// TIA Portal project "Cuối kì" (V16)

(* hardware
DEVICE "S7-1200 station_1"  S7-1200 Station
   slot 0: "Rack_0"  S7-1200 Rack  Rack  V1.0
   slot 1: "PLC_1"  CPU 1212C DC/DC/DC  6ES7 212-1AE40-0XB0  V4.4
*)

// ===== PLC "PLC_1"  CPU 1212C DC/DC/DC =====

VAR_GLOBAL   // PLC tag table "Default tag table"
   "Clock_Byte" AT %MB21 : Byte;
   "Clock_10Hz" AT %M21.0 : Bool;
   "Clock_5Hz" AT %M21.1 : Bool;
   "Clock_2.5Hz" AT %M21.2 : Bool;
   "Clock_2Hz" AT %M21.3 : Bool;
   "Clock_1.25Hz" AT %M21.4 : Bool;
   "Clock_1Hz" AT %M21.5 : Bool;
   "Clock_0.625Hz" AT %M21.6 : Bool;
   "Clock_0.5Hz" AT %M21.7 : Bool;
   "iStart" AT %M0.0 : Bool;
   "iStop" AT %M0.1 : Bool;
   "enableSystem" AT %M0.2 : Bool;
   "mEnableXiloRice" AT %M0.3 : Bool;
   "mEnableXiloCorn" AT %M0.4 : Bool;
   "mEnableXiloManioc" AT %M0.5 : Bool;
   "mEnableXiloBean" AT %M0.6 : Bool;
   "mEnableXiloFish" AT %M0.7 : Bool;
   "mLetOutRice" AT %M1.0 : Bool;
   "mLetOutCorn" AT %M1.1 : Bool;
   "mLetOutManioc" AT %M1.2 : Bool;
   "mLetOutBean" AT %M1.3 : Bool;
   "mLetOutFish" AT %M1.4 : Bool;
   "mLightRice" AT %M1.5 : Bool;
   "mLightCorn" AT %M1.6 : Bool;
   "mLightManioc" AT %M1.7 : Bool;
   "mLightBean" AT %M2.0 : Bool;
   "mLightFish" AT %M2.1 : Bool;
   "iResetCTU" AT %M2.2 : Bool;
   "oXilo1" AT %Q0.0 : Bool;
   "oXilo2" AT %Q0.1 : Bool;
   "oXilo3" AT %Q0.2 : Bool;
   "oXilo4" AT %Q0.3 : Bool;
   "oXilo5" AT %Q0.4 : Bool;
   "oXilo6" AT %Q0.5 : Bool;
   "oXilo7" AT %Q0.6 : Bool;
   "oXilo8" AT %Q0.7 : Bool;
   "oXilo9" AT %Q1.0 : Bool;
   "oXilo10" AT %Q1.1 : Bool;
   "oXilo11" AT %Q1.2 : Bool;
   "oXilo12" AT %Q1.3 : Bool;
   "oXilo13" AT %Q1.4 : Bool;
   "oXilo14" AT %Q1.5 : Bool;
   "oXilo15" AT %Q1.6 : Bool;
   "oXilo16" AT %Q1.7 : Bool;
   "mLetOutScale" AT %M2.3 : Bool;
   "iSensor1" AT %M2.4 : Bool;
   "iSensorHigh2" AT %M2.5 : Bool;
   "iSensorLow2" AT %M2.6 : Bool;
   "oValve1" AT %Q2.0 : Bool;
   "oValve2" AT %Q2.1 : Bool;
   "iResetCTD" AT %M2.7 : Bool;
   "mTank" AT %M3.0 : Bool;
   "Tag_3" AT %M100.1 : Bool;
   "Tag_4" AT %M100.2 : Bool;
   "oMix" AT %Q2.2 : Bool;
   "iContinue" AT %M3.1 : Bool;
   "Continue" AT %M3.2 : Bool;
   "oValve3" AT %Q2.3 : Bool;
   "iSensor3" AT %M3.4 : Bool;
   "Hold11" AT %M3.6 : Bool;
   "Hold21" AT %M3.7 : Bool;
   "Hold31" AT %M4.0 : Bool;
   "Hold41" AT %M4.1 : Bool;
   "Hold51" AT %M4.2 : Bool;
   "Reset" AT %M4.3 : Bool;
   "Hold12" AT %M4.4 : Bool;
   "Hold13" AT %M4.5 : Bool;
   "Hold14" AT %M4.6 : Bool;
   "Hold15" AT %M4.7 : Bool;
   "Hold22" AT %M5.0 : Bool;
   "Hold23" AT %M5.1 : Bool;
   "Hold24" AT %M5.2 : Bool;
   "Hold25" AT %M5.3 : Bool;
   "Hold32" AT %M5.4 : Bool;
   "Hold33" AT %M5.5 : Bool;
   "Hold34" AT %M5.6 : Bool;
   "Hold35" AT %M5.7 : Bool;
   "Hold42" AT %M6.0 : Bool;
   "Hold52" AT %M6.1 : Bool;
   "Tag_1" AT %MW1 : Int;
   "Tag_2" AT %MW2 : Int;
   "Tag_5" AT %MW3 : Int;
   "Tag_6" AT %MW4 : Int;
   "Tag_7" AT %MW5 : Int;
   "Tag_8" AT %MW6 : Int;
   "Tag_9" AT %MW7 : Int;
   "Tag_10" AT %MW8 : Int;
   "Tag_11" AT %MW9 : Int;
   "Tag_12" AT %MW10 : Int;
   "Tag_13" AT %MW11 : Int;
   "Tag_14" AT %MW12 : Int;
   "Tag_15" AT %MW13 : Int;
   "Tag_16" AT %MW14 : Int;
   "Tag_17" AT %MW15 : Int;
   "Tag_18" AT %MW16 : Int;
   "Tag_19" AT %MW17 : Int;
   "Tag_20" AT %MW18 : Int;
   "Tag_21" AT %MD1 : Time;
   "oSensor1" AT %M6.2 : Bool;
   "oSensor3" AT %M6.3 : Bool;
END_VAR

DATA_BLOCK "Mass"   // DB1
{ S7_Optimized_Access := 'FALSE' }
VERSION : 0.1
   VAR
      Rice : Int := 5;
      Corn : Int := 5;
      Manioc : Int := 5;
      Bean : Int := 5;
      Fish : Int := 5;
   END_VAR
BEGIN
END_DATA_BLOCK

DATA_BLOCK "TimeMix"   // DB2
{ S7_Optimized_Access := 'FALSE' }
VERSION : 0.1
   VAR
      "Time" : Time := T#40S;
   END_VAR
BEGIN
END_DATA_BLOCK

DATA_BLOCK "Sum"   // DB22
{ S7_Optimized_Access := 'FALSE' }
VERSION : 0.1
   VAR
      Rice : Int := 60;
      Corn : Int := 50;
      Manioc : Int := 60;
      Bean : Int := 30;
      Fish : Int := 60;
      Sum1 : Int := 100;
      Sum2 : Int := 200;
   END_VAR
BEGIN
END_DATA_BLOCK

DATA_BLOCK "Weight"   // DB23
{ S7_Optimized_Access := 'FALSE' }
VERSION : 0.1
   VAR
      Xilo1 : Int;
      Xilo2 : Int;
      Xilo3 : Int;
      Xilo4 : Int;
      Xilo5 : Int;
      Xilo6 : Int;
      Xilo7 : Int;
      Xilo8 : Int;
      Xilo9 : Int;
      Xilo10 : Int;
      Xilo11 : Int;
      Xilo12 : Int;
      Xilo13 : Int;
      Xilo14 : Int;
      Xilo15 : Int;
      Xilo16 : Int;
      Sum1 : Int;
      Sum2 : Int;
   END_VAR
BEGIN
END_DATA_BLOCK

DATA_BLOCK "ADD"   // DB24
{ S7_Optimized_Access := 'FALSE' }
VERSION : 0.1
   VAR
      ScaleSum1 : Int;
      ScaleSum2 : Int;
   END_VAR
BEGIN
END_DATA_BLOCK

// folder: System blocks/Program resources

DATA_BLOCK "Scale8"   // DB3
{ S7_Optimized_Access := 'TRUE' }
AUTHOR : Simatic
FAMILY : IEC
NAME : CNTR
VERSION : 1.0
// stored: InstanceOfName IEC_COUNTER
"IEC_COUNTER"
BEGIN
END_DATA_BLOCK

DATA_BLOCK "Scale9"   // DB4
{ S7_Optimized_Access := 'TRUE' }
AUTHOR : Simatic
FAMILY : IEC
NAME : CNTR
VERSION : 1.0
// stored: InstanceOfName IEC_COUNTER
"IEC_COUNTER"
BEGIN
END_DATA_BLOCK

DATA_BLOCK "Scale4"   // DB5
{ S7_Optimized_Access := 'TRUE' }
AUTHOR : Simatic
FAMILY : IEC
NAME : CNTR
VERSION : 1.0
// stored: InstanceOfName IEC_COUNTER
"IEC_COUNTER"
BEGIN
END_DATA_BLOCK

DATA_BLOCK "Scale5"   // DB6
{ S7_Optimized_Access := 'TRUE' }
AUTHOR : Simatic
FAMILY : IEC
NAME : CNTR
VERSION : 1.0
// stored: InstanceOfName IEC_COUNTER
"IEC_COUNTER"
BEGIN
END_DATA_BLOCK

DATA_BLOCK "Scale6"   // DB7
{ S7_Optimized_Access := 'TRUE' }
AUTHOR : Simatic
FAMILY : IEC
NAME : CNTR
VERSION : 1.0
// stored: InstanceOfName IEC_COUNTER
"IEC_COUNTER"
BEGIN
END_DATA_BLOCK

DATA_BLOCK "Scale7"   // DB8
{ S7_Optimized_Access := 'TRUE' }
AUTHOR : Simatic
FAMILY : IEC
NAME : CNTR
VERSION : 1.0
// stored: InstanceOfName IEC_COUNTER
"IEC_COUNTER"
BEGIN
END_DATA_BLOCK

DATA_BLOCK "Scale1"   // DB9
{ S7_Optimized_Access := 'TRUE' }
AUTHOR : Simatic
FAMILY : IEC
NAME : CNTR
VERSION : 1.0
// stored: InstanceOfName IEC_COUNTER
"IEC_COUNTER"
BEGIN
END_DATA_BLOCK

DATA_BLOCK "Scale2"   // DB10
{ S7_Optimized_Access := 'TRUE' }
AUTHOR : Simatic
FAMILY : IEC
NAME : CNTR
VERSION : 1.0
// stored: InstanceOfName IEC_COUNTER
"IEC_COUNTER"
BEGIN
END_DATA_BLOCK

DATA_BLOCK "Scale3"   // DB11
{ S7_Optimized_Access := 'TRUE' }
AUTHOR : Simatic
FAMILY : IEC
NAME : CNTR
VERSION : 1.0
// stored: InstanceOfName IEC_COUNTER
"IEC_COUNTER"
BEGIN
END_DATA_BLOCK

DATA_BLOCK "Scale10"   // DB12
{ S7_Optimized_Access := 'TRUE' }
AUTHOR : Simatic
FAMILY : IEC
NAME : CNTR
VERSION : 1.0
// stored: InstanceOfName IEC_COUNTER
"IEC_COUNTER"
BEGIN
END_DATA_BLOCK

DATA_BLOCK "Scale11"   // DB13
{ S7_Optimized_Access := 'TRUE' }
AUTHOR : Simatic
FAMILY : IEC
NAME : CNTR
VERSION : 1.0
// stored: InstanceOfName IEC_COUNTER
"IEC_COUNTER"
BEGIN
END_DATA_BLOCK

DATA_BLOCK "Scale12"   // DB14
{ S7_Optimized_Access := 'TRUE' }
AUTHOR : Simatic
FAMILY : IEC
NAME : CNTR
VERSION : 1.0
// stored: InstanceOfName IEC_COUNTER
"IEC_COUNTER"
BEGIN
END_DATA_BLOCK

DATA_BLOCK "Scale13"   // DB15
{ S7_Optimized_Access := 'TRUE' }
AUTHOR : Simatic
FAMILY : IEC
NAME : CNTR
VERSION : 1.0
// stored: InstanceOfName IEC_COUNTER
"IEC_COUNTER"
BEGIN
END_DATA_BLOCK

DATA_BLOCK "Scale14"   // DB16
{ S7_Optimized_Access := 'TRUE' }
AUTHOR : Simatic
FAMILY : IEC
NAME : CNTR
VERSION : 1.0
// stored: InstanceOfName IEC_COUNTER
"IEC_COUNTER"
BEGIN
END_DATA_BLOCK

DATA_BLOCK "Scale15"   // DB17
{ S7_Optimized_Access := 'TRUE' }
AUTHOR : Simatic
FAMILY : IEC
NAME : CNTR
VERSION : 1.0
// stored: InstanceOfName IEC_COUNTER
"IEC_COUNTER"
BEGIN
END_DATA_BLOCK

DATA_BLOCK "Scale16"   // DB18
{ S7_Optimized_Access := 'TRUE' }
AUTHOR : Simatic
FAMILY : IEC
NAME : CNTR
VERSION : 1.0
// stored: InstanceOfName IEC_COUNTER
"IEC_COUNTER"
BEGIN
END_DATA_BLOCK

DATA_BLOCK "ScaleSum"   // DB19
{ S7_Optimized_Access := 'TRUE' }
AUTHOR : Simatic
FAMILY : IEC
NAME : CNTR
VERSION : 1.0
// stored: InstanceOfName IEC_COUNTER
"IEC_COUNTER"
BEGIN
END_DATA_BLOCK

DATA_BLOCK "Time"   // DB20
{ S7_Optimized_Access := 'TRUE' }
AUTHOR : Simatic
FAMILY : IEC
NAME : IEC_TMR
VERSION : 1.0
// stored: InstanceOfName IEC_TIMER
"IEC_TIMER"
BEGIN
END_DATA_BLOCK

DATA_BLOCK "ScaleSum2"   // DB21
{ S7_Optimized_Access := 'TRUE' }
AUTHOR : Simatic
FAMILY : IEC
NAME : CNTR
VERSION : 1.0
// stored: InstanceOfName IEC_COUNTER
"IEC_COUNTER"
BEGIN
END_DATA_BLOCK

// folder: (top level)

ORGANIZATION_BLOCK "Main"   // OB1, LAD, ProgramCycle
TITLE = "Main Program Sweep (Cycle)"
{ S7_Optimized_Access := 'TRUE' }
VERSION : 0.1
   VAR_INPUT
      Initial_Call : Bool;   // Initial call of this OB
      Remanence : Bool;   // =True, if remanent data are available
   END_VAR
   VAR_TEMP   // added for the SCL form of the ladder/FBD networks
      _w1 : Bool;
      _w2 : Bool;
      _w3 : Bool;
   END_VAR
BEGIN

REGION Network 1: Open/Close System
   // Bắt đầu + đóng + tiếp tục + reset counter
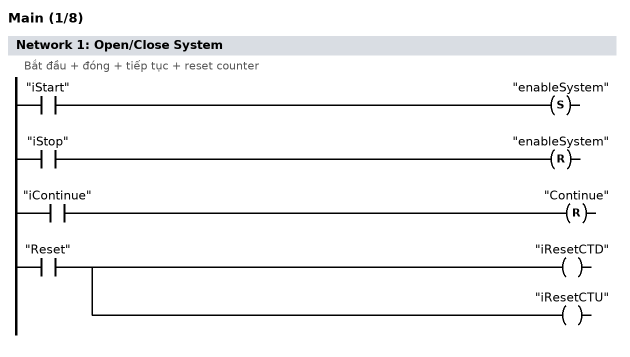
   RUNG wire#powerrail
      Contact( "iStart" )
      S_Coil( "enableSystem" )
   END_RUNG
   RUNG wire#powerrail
      Contact( "iStop" )
      R_Coil( "enableSystem" )
   END_RUNG
   RUNG wire#powerrail
      Contact( "iContinue" )
      R_Coil( "Continue" )
   END_RUNG
   RUNG wire#powerrail
      Contact( "Reset" )
      wire#w1
      Coil( "iResetCTD" )
   END_RUNG
   RUNG wire#w1
      Coil( "iResetCTU" )
   END_RUNG
   // the same network as SCL:
   IF "iStart" THEN "enableSystem" := TRUE; END_IF;
   IF "iStop" THEN "enableSystem" := FALSE; END_IF;
   IF "iContinue" THEN "Continue" := FALSE; END_IF;
   "iResetCTD" := "Reset";
   "iResetCTU" := "Reset";
END_REGION

REGION Network 2: So sánh khối lượng
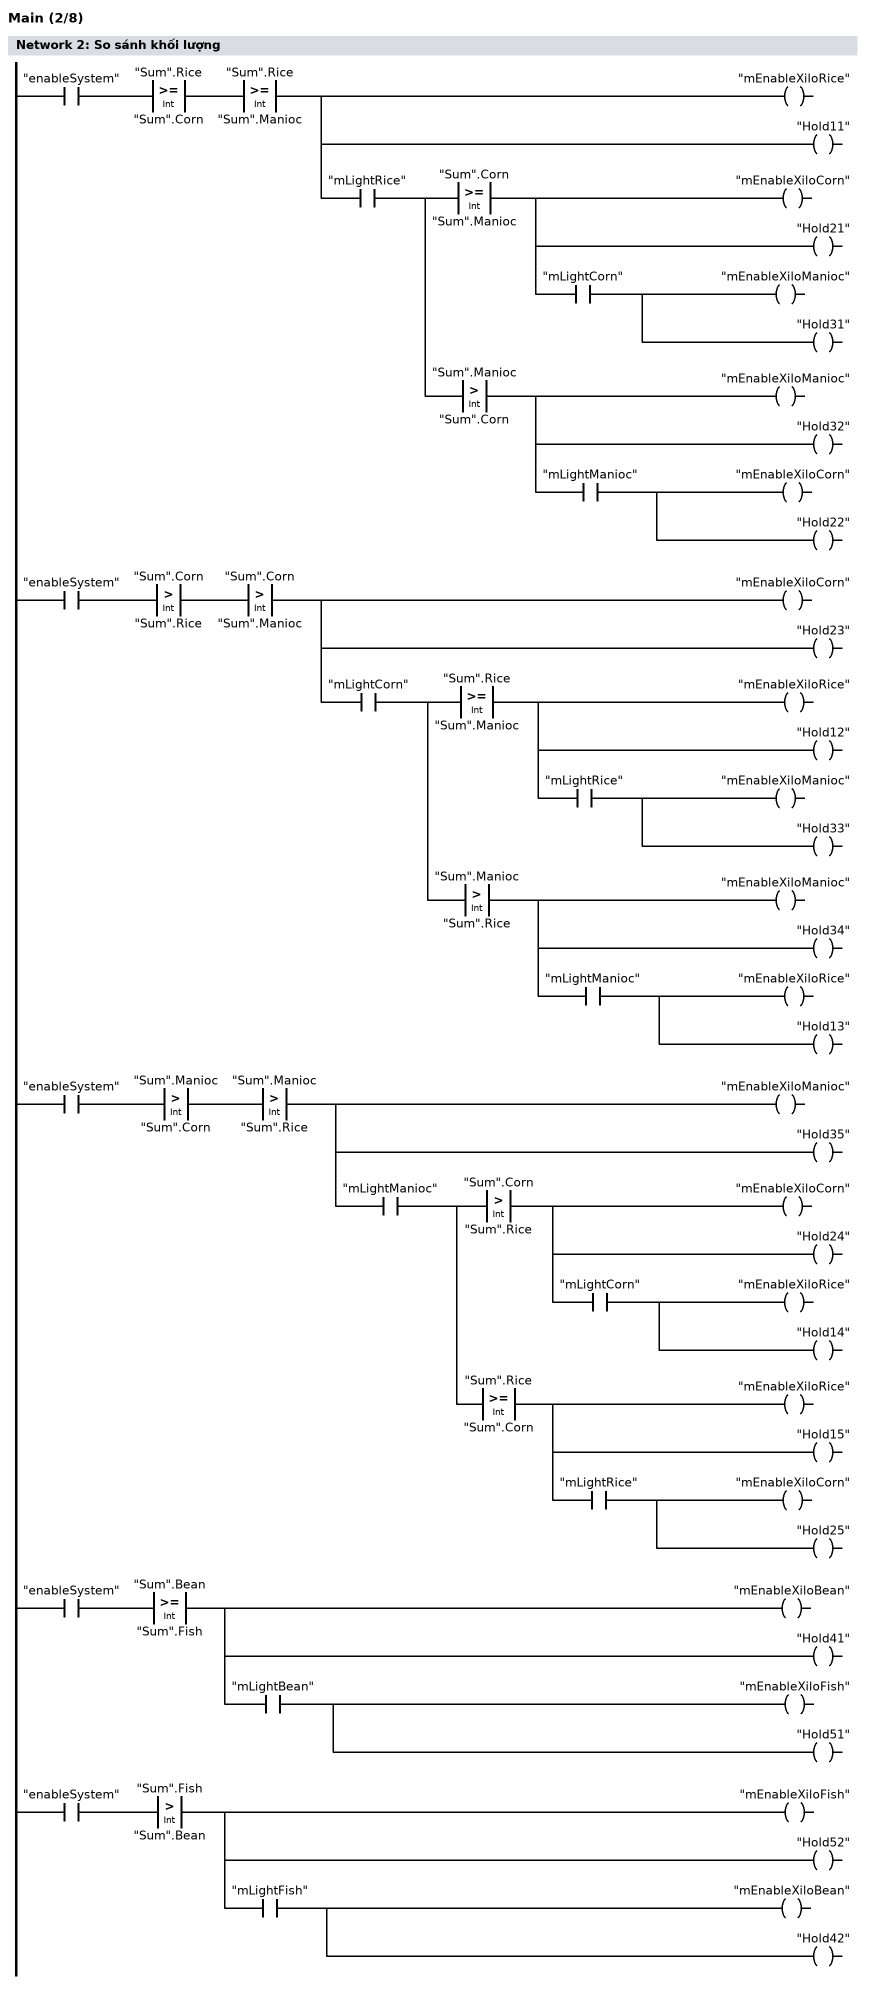
   RUNG wire#powerrail
      Contact( "enableSystem" )
      { S7_Templates := "SrcType := Int" } GE_Contact(in1 := "Sum".Rice, in2 := "Sum".Corn)
      { S7_Templates := "SrcType := Int" } GE_Contact(in1 := "Sum".Rice, in2 := "Sum".Manioc)
      wire#w1
      Coil( "mEnableXiloRice" )
   END_RUNG
   RUNG wire#w1
      Coil( "Hold11" )
   END_RUNG
   RUNG wire#w1
      Contact( "mLightRice" )
      wire#w2
      { S7_Templates := "SrcType := Int" } GE_Contact(in1 := "Sum".Corn, in2 := "Sum".Manioc)
      wire#w3
      Coil( "mEnableXiloCorn" )
   END_RUNG
   RUNG wire#w3
      Coil( "Hold21" )
   END_RUNG
   RUNG wire#w3
      Contact( "mLightCorn" )
      wire#w4
      Coil( "mEnableXiloManioc" )
   END_RUNG
   RUNG wire#w4
      Coil( "Hold31" )
   END_RUNG
   RUNG wire#w2
      { S7_Templates := "SrcType := Int" } GT_Contact(in1 := "Sum".Manioc, in2 := "Sum".Corn)
      wire#w5
      Coil( "mEnableXiloManioc" )
   END_RUNG
   RUNG wire#w5
      Coil( "Hold32" )
   END_RUNG
   RUNG wire#w5
      Contact( "mLightManioc" )
      wire#w6
      Coil( "mEnableXiloCorn" )
   END_RUNG
   RUNG wire#w6
      Coil( "Hold22" )
   END_RUNG
   RUNG wire#powerrail
      Contact( "enableSystem" )
      { S7_Templates := "SrcType := Int" } GT_Contact(in1 := "Sum".Corn, in2 := "Sum".Rice)
      { S7_Templates := "SrcType := Int" } GT_Contact(in1 := "Sum".Corn, in2 := "Sum".Manioc)
      wire#w7
      Coil( "mEnableXiloCorn" )
   END_RUNG
   RUNG wire#w7
      Coil( "Hold23" )
   END_RUNG
   RUNG wire#w7
      Contact( "mLightCorn" )
      wire#w8
      { S7_Templates := "SrcType := Int" } GE_Contact(in1 := "Sum".Rice, in2 := "Sum".Manioc)
      wire#w9
      Coil( "mEnableXiloRice" )
   END_RUNG
   RUNG wire#w9
      Coil( "Hold12" )
   END_RUNG
   RUNG wire#w9
      Contact( "mLightRice" )
      wire#w10
      Coil( "mEnableXiloManioc" )
   END_RUNG
   RUNG wire#w10
      Coil( "Hold33" )
   END_RUNG
   RUNG wire#w8
      { S7_Templates := "SrcType := Int" } GT_Contact(in1 := "Sum".Manioc, in2 := "Sum".Rice)
      wire#w11
      Coil( "mEnableXiloManioc" )
   END_RUNG
   RUNG wire#w11
      Coil( "Hold34" )
   END_RUNG
   RUNG wire#w11
      Contact( "mLightManioc" )
      wire#w12
      Coil( "mEnableXiloRice" )
   END_RUNG
   RUNG wire#w12
      Coil( "Hold13" )
   END_RUNG
   RUNG wire#powerrail
      Contact( "enableSystem" )
      { S7_Templates := "SrcType := Int" } GT_Contact(in1 := "Sum".Manioc, in2 := "Sum".Corn)
      { S7_Templates := "SrcType := Int" } GT_Contact(in1 := "Sum".Manioc, in2 := "Sum".Rice)
      wire#w13
      Coil( "mEnableXiloManioc" )
   END_RUNG
   RUNG wire#w13
      Coil( "Hold35" )
   END_RUNG
   RUNG wire#w13
      Contact( "mLightManioc" )
      wire#w14
      { S7_Templates := "SrcType := Int" } GT_Contact(in1 := "Sum".Corn, in2 := "Sum".Rice)
      wire#w15
      Coil( "mEnableXiloCorn" )
   END_RUNG
   RUNG wire#w15
      Coil( "Hold24" )
   END_RUNG
   RUNG wire#w15
      Contact( "mLightCorn" )
      wire#w16
      Coil( "mEnableXiloRice" )
   END_RUNG
   RUNG wire#w16
      Coil( "Hold14" )
   END_RUNG
   RUNG wire#w14
      { S7_Templates := "SrcType := Int" } GE_Contact(in1 := "Sum".Rice, in2 := "Sum".Corn)
      wire#w17
      Coil( "mEnableXiloRice" )
   END_RUNG
   RUNG wire#w17
      Coil( "Hold15" )
   END_RUNG
   RUNG wire#w17
      Contact( "mLightRice" )
      wire#w18
      Coil( "mEnableXiloCorn" )
   END_RUNG
   RUNG wire#w18
      Coil( "Hold25" )
   END_RUNG
   RUNG wire#powerrail
      Contact( "enableSystem" )
      { S7_Templates := "SrcType := Int" } GE_Contact(in1 := "Sum".Bean, in2 := "Sum".Fish)
      wire#w19
      Coil( "mEnableXiloBean" )
   END_RUNG
   RUNG wire#w19
      Coil( "Hold41" )
   END_RUNG
   RUNG wire#w19
      Contact( "mLightBean" )
      wire#w20
      Coil( "mEnableXiloFish" )
   END_RUNG
   RUNG wire#w20
      Coil( "Hold51" )
   END_RUNG
   RUNG wire#powerrail
      Contact( "enableSystem" )
      { S7_Templates := "SrcType := Int" } GT_Contact(in1 := "Sum".Fish, in2 := "Sum".Bean)
      wire#w21
      Coil( "mEnableXiloFish" )
   END_RUNG
   RUNG wire#w21
      Coil( "Hold52" )
   END_RUNG
   RUNG wire#w21
      Contact( "mLightFish" )
      wire#w22
      Coil( "mEnableXiloBean" )
   END_RUNG
   RUNG wire#w22
      Coil( "Hold42" )
   END_RUNG
   // the same network as SCL:
   "mEnableXiloRice" := "enableSystem" AND ("Sum".Rice >= "Sum".Corn) AND ("Sum".Rice >= "Sum".Manioc);
   "Hold11" := "mEnableXiloRice";
   #_w1 := "mEnableXiloRice" AND "mLightRice";
   "mEnableXiloCorn" := #_w1 AND ("Sum".Corn >= "Sum".Manioc);
   "Hold21" := "mEnableXiloCorn";
   "mEnableXiloManioc" := "mEnableXiloCorn" AND "mLightCorn";
   "Hold31" := "mEnableXiloManioc";
   "mEnableXiloManioc" := #_w1 AND ("Sum".Manioc > "Sum".Corn);
   "Hold32" := "mEnableXiloManioc";
   "mEnableXiloCorn" := "mEnableXiloManioc" AND "mLightManioc";
   "Hold22" := "mEnableXiloCorn";
   "mEnableXiloCorn" := "enableSystem" AND ("Sum".Corn > "Sum".Rice) AND ("Sum".Corn > "Sum".Manioc);
   "Hold23" := "mEnableXiloCorn";
   #_w2 := "mEnableXiloCorn" AND "mLightCorn";
   "mEnableXiloRice" := #_w2 AND ("Sum".Rice >= "Sum".Manioc);
   "Hold12" := "mEnableXiloRice";
   "mEnableXiloManioc" := "mEnableXiloRice" AND "mLightRice";
   "Hold33" := "mEnableXiloManioc";
   "mEnableXiloManioc" := #_w2 AND ("Sum".Manioc > "Sum".Rice);
   "Hold34" := "mEnableXiloManioc";
   "mEnableXiloRice" := "mEnableXiloManioc" AND "mLightManioc";
   "Hold13" := "mEnableXiloRice";
   "mEnableXiloManioc" := "enableSystem" AND ("Sum".Manioc > "Sum".Corn) AND ("Sum".Manioc > "Sum".Rice);
   "Hold35" := "mEnableXiloManioc";
   #_w3 := "mEnableXiloManioc" AND "mLightManioc";
   "mEnableXiloCorn" := #_w3 AND ("Sum".Corn > "Sum".Rice);
   "Hold24" := "mEnableXiloCorn";
   "mEnableXiloRice" := "mEnableXiloCorn" AND "mLightCorn";
   "Hold14" := "mEnableXiloRice";
   "mEnableXiloRice" := #_w3 AND ("Sum".Rice >= "Sum".Corn);
   "Hold15" := "mEnableXiloRice";
   "mEnableXiloCorn" := "mEnableXiloRice" AND "mLightRice";
   "Hold25" := "mEnableXiloCorn";
   "mEnableXiloBean" := "enableSystem" AND ("Sum".Bean >= "Sum".Fish);
   "Hold41" := "mEnableXiloBean";
   "mEnableXiloFish" := "mEnableXiloBean" AND "mLightBean";
   "Hold51" := "mEnableXiloFish";
   "mEnableXiloFish" := "enableSystem" AND ("Sum".Fish > "Sum".Bean);
   "Hold52" := "mEnableXiloFish";
   "mEnableXiloBean" := "mEnableXiloFish" AND "mLightFish";
   "Hold42" := "mEnableXiloBean";
END_REGION

REGION Network 3: Mở nguồn các xilo
   // Mở nguồn các xilo
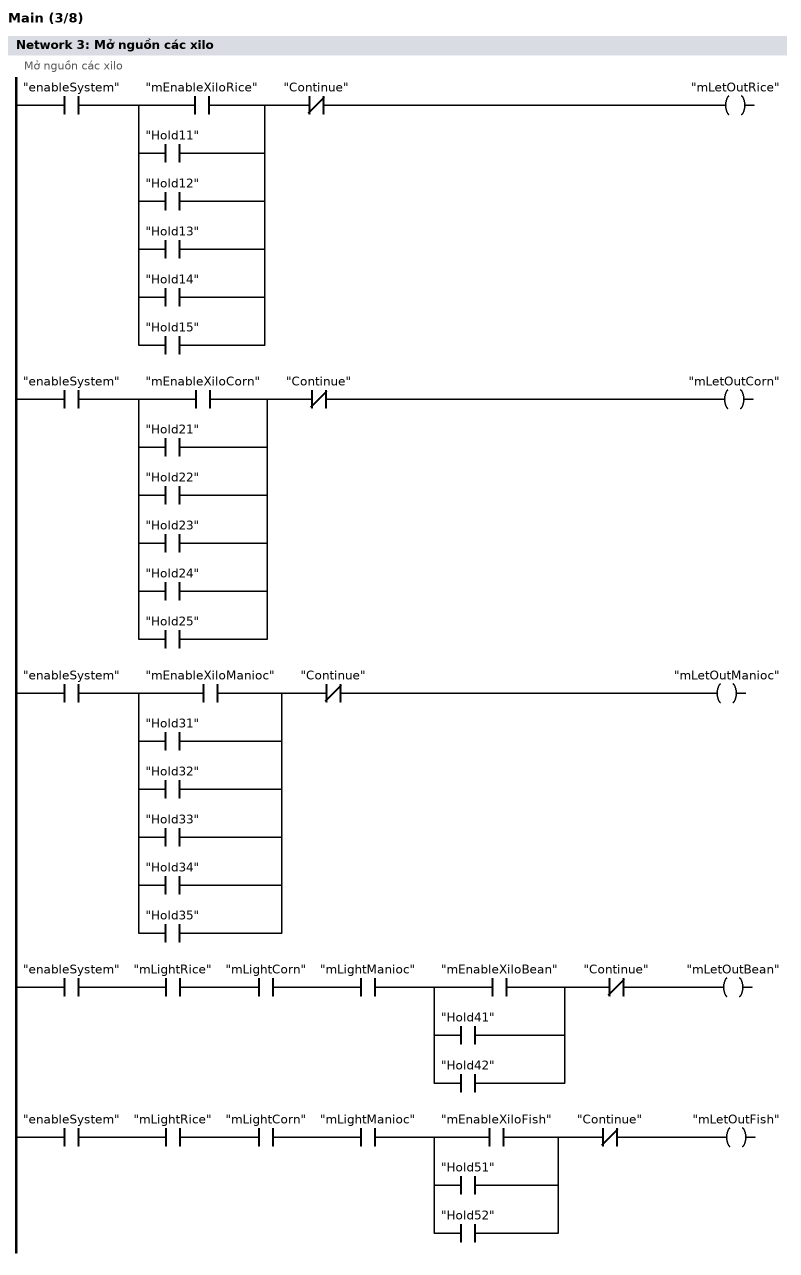
   RUNG wire#powerrail
      Contact( "enableSystem" )
      wire#w1
      Contact( "mEnableXiloRice" )
      wire#w2
      I_Contact( "Continue" )
      Coil( "mLetOutRice" )
   END_RUNG
   RUNG wire#w1
      Contact( "Hold11" )
   END_RUNG wire#w2
   RUNG wire#w1
      Contact( "Hold12" )
   END_RUNG wire#w2
   RUNG wire#w1
      Contact( "Hold13" )
   END_RUNG wire#w2
   RUNG wire#w1
      Contact( "Hold14" )
   END_RUNG wire#w2
   RUNG wire#w1
      Contact( "Hold15" )
   END_RUNG wire#w2
   RUNG wire#powerrail
      Contact( "enableSystem" )
      wire#w3
      Contact( "mEnableXiloCorn" )
      wire#w4
      I_Contact( "Continue" )
      Coil( "mLetOutCorn" )
   END_RUNG
   RUNG wire#w3
      Contact( "Hold21" )
   END_RUNG wire#w4
   RUNG wire#w3
      Contact( "Hold22" )
   END_RUNG wire#w4
   RUNG wire#w3
      Contact( "Hold23" )
   END_RUNG wire#w4
   RUNG wire#w3
      Contact( "Hold24" )
   END_RUNG wire#w4
   RUNG wire#w3
      Contact( "Hold25" )
   END_RUNG wire#w4
   RUNG wire#powerrail
      Contact( "enableSystem" )
      wire#w5
      Contact( "mEnableXiloManioc" )
      wire#w6
      I_Contact( "Continue" )
      Coil( "mLetOutManioc" )
   END_RUNG
   RUNG wire#w5
      Contact( "Hold31" )
   END_RUNG wire#w6
   RUNG wire#w5
      Contact( "Hold32" )
   END_RUNG wire#w6
   RUNG wire#w5
      Contact( "Hold33" )
   END_RUNG wire#w6
   RUNG wire#w5
      Contact( "Hold34" )
   END_RUNG wire#w6
   RUNG wire#w5
      Contact( "Hold35" )
   END_RUNG wire#w6
   RUNG wire#powerrail
      Contact( "enableSystem" )
      Contact( "mLightRice" )
      Contact( "mLightCorn" )
      Contact( "mLightManioc" )
      wire#w7
      Contact( "mEnableXiloBean" )
      wire#w8
      I_Contact( "Continue" )
      Coil( "mLetOutBean" )
   END_RUNG
   RUNG wire#w7
      Contact( "Hold41" )
   END_RUNG wire#w8
   RUNG wire#w7
      Contact( "Hold42" )
   END_RUNG wire#w8
   RUNG wire#powerrail
      Contact( "enableSystem" )
      Contact( "mLightRice" )
      Contact( "mLightCorn" )
      Contact( "mLightManioc" )
      wire#w9
      Contact( "mEnableXiloFish" )
      wire#w10
      I_Contact( "Continue" )
      Coil( "mLetOutFish" )
   END_RUNG
   RUNG wire#w9
      Contact( "Hold51" )
   END_RUNG wire#w10
   RUNG wire#w9
      Contact( "Hold52" )
   END_RUNG wire#w10
   // the same network as SCL:
   "mLetOutRice" := "enableSystem" AND ("mEnableXiloRice" OR "Hold11" OR "Hold12" OR "Hold13" OR "Hold14" OR "Hold15") AND NOT "Continue";
   "mLetOutCorn" := "enableSystem" AND ("mEnableXiloCorn" OR "Hold21" OR "Hold22" OR "Hold23" OR "Hold24" OR "Hold25") AND NOT "Continue";
   "mLetOutManioc" := "enableSystem" AND ("mEnableXiloManioc" OR "Hold31" OR "Hold32" OR "Hold33" OR "Hold34" OR "Hold35") AND NOT "Continue";
   "mLetOutBean" := "enableSystem" AND "mLightRice" AND "mLightCorn" AND "mLightManioc" AND ("mEnableXiloBean" OR "Hold41" OR "Hold42") AND NOT "Continue";
   "mLetOutFish" := "enableSystem" AND "mLightRice" AND "mLightCorn" AND "mLightManioc" AND ("mEnableXiloFish" OR "Hold51" OR "Hold52") AND NOT "Continue";
END_REGION

REGION Network 4: xả xilo 1,2,3 (bột gạo)
   // xả xilo 1,2,3 (bột gạo)
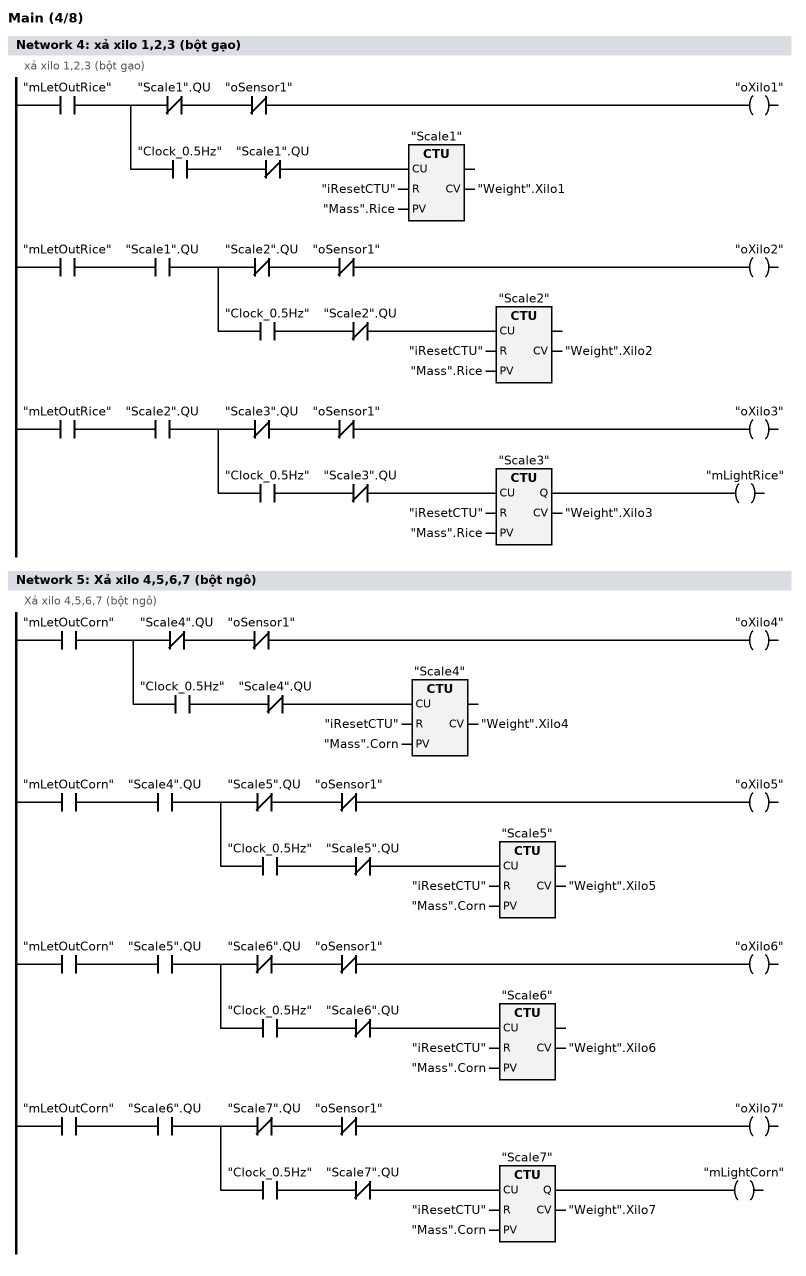
   "oXilo1" := "mLetOutRice" AND NOT "Scale1".QU AND NOT "oSensor1";
   "Scale1".CTU(CU := "mLetOutRice" AND "Clock_0.5Hz" AND NOT "Scale1".QU,
                R := "iResetCTU",
                PV := "Mass".Rice,
                CV => "Weight".Xilo1);
   #_w1 := "mLetOutRice" AND "Scale1".QU;
   "oXilo2" := #_w1 AND NOT "Scale2".QU AND NOT "oSensor1";
   "Scale2".CTU(CU := #_w1 AND "Clock_0.5Hz" AND NOT "Scale2".QU,
                R := "iResetCTU",
                PV := "Mass".Rice,
                CV => "Weight".Xilo2);
   #_w2 := "mLetOutRice" AND "Scale2".QU;
   "oXilo3" := #_w2 AND NOT "Scale3".QU AND NOT "oSensor1";
   "Scale3".CTU(CU := #_w2 AND "Clock_0.5Hz" AND NOT "Scale3".QU,
                R := "iResetCTU",
                PV := "Mass".Rice,
                CV => "Weight".Xilo3);
   "mLightRice" := "Scale3".Q;
END_REGION

REGION Network 5: Xả xilo 4,5,6,7 (bột ngô)
   // Xả xilo 4,5,6,7 (bột ngô)
   "oXilo4" := "mLetOutCorn" AND NOT "Scale4".QU AND NOT "oSensor1";
   "Scale4".CTU(CU := "mLetOutCorn" AND "Clock_0.5Hz" AND NOT "Scale4".QU,
                R := "iResetCTU",
                PV := "Mass".Corn,
                CV => "Weight".Xilo4);
   #_w1 := "mLetOutCorn" AND "Scale4".QU;
   "oXilo5" := #_w1 AND NOT "Scale5".QU AND NOT "oSensor1";
   "Scale5".CTU(CU := #_w1 AND "Clock_0.5Hz" AND NOT "Scale5".QU,
                R := "iResetCTU",
                PV := "Mass".Corn,
                CV => "Weight".Xilo5);
   #_w2 := "mLetOutCorn" AND "Scale5".QU;
   "oXilo6" := #_w2 AND NOT "Scale6".QU AND NOT "oSensor1";
   "Scale6".CTU(CU := #_w2 AND "Clock_0.5Hz" AND NOT "Scale6".QU,
                R := "iResetCTU",
                PV := "Mass".Corn,
                CV => "Weight".Xilo6);
   #_w3 := "mLetOutCorn" AND "Scale6".QU;
   "oXilo7" := #_w3 AND NOT "Scale7".QU AND NOT "oSensor1";
   "Scale7".CTU(CU := #_w3 AND "Clock_0.5Hz" AND NOT "Scale7".QU,
                R := "iResetCTU",
                PV := "Mass".Corn,
                CV => "Weight".Xilo7);
   "mLightCorn" := "Scale7".Q;
END_REGION

REGION Network 6: Xả xilo 8,9 ( bột sắn )
   // Xả xilo 8,9 ( bột sắn )
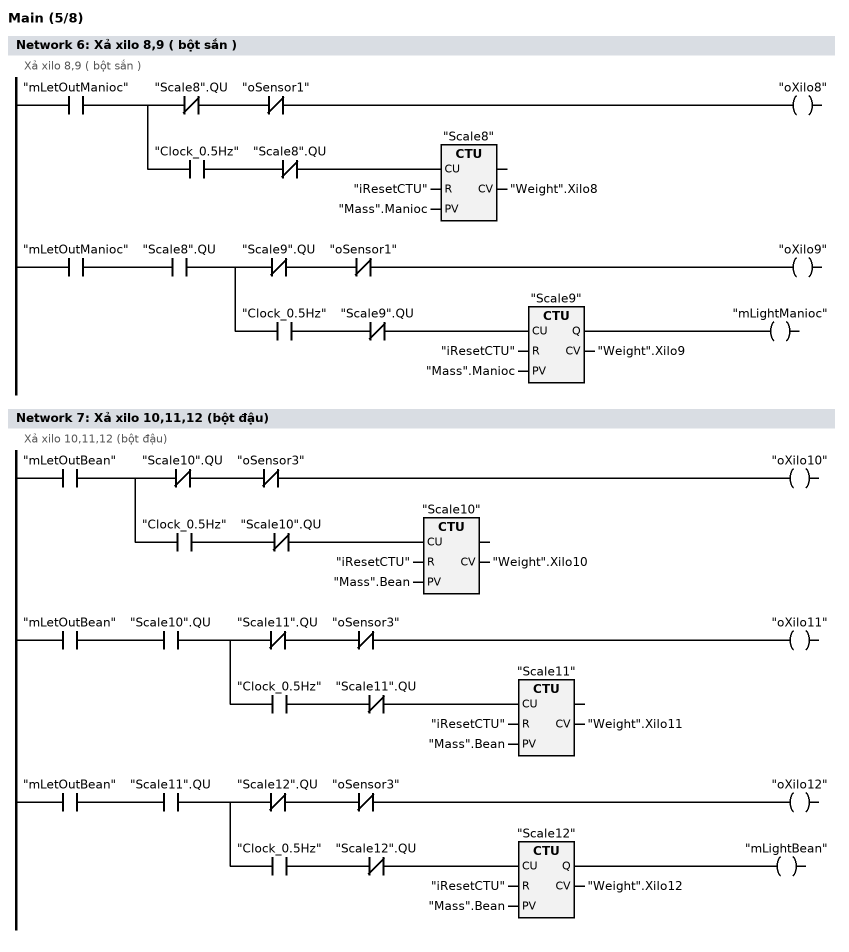
   "oXilo8" := "mLetOutManioc" AND NOT "Scale8".QU AND NOT "oSensor1";
   "Scale8".CTU(CU := "mLetOutManioc" AND "Clock_0.5Hz" AND NOT "Scale8".QU,
                R := "iResetCTU",
                PV := "Mass".Manioc,
                CV => "Weight".Xilo8);
   #_w1 := "mLetOutManioc" AND "Scale8".QU;
   "oXilo9" := #_w1 AND NOT "Scale9".QU AND NOT "oSensor1";
   "Scale9".CTU(CU := #_w1 AND "Clock_0.5Hz" AND NOT "Scale9".QU,
                R := "iResetCTU",
                PV := "Mass".Manioc,
                CV => "Weight".Xilo9);
   "mLightManioc" := "Scale9".Q;
END_REGION

REGION Network 7: Xả xilo 10,11,12 (bột đậu)
   // Xả xilo 10,11,12 (bột đậu)
   "oXilo10" := "mLetOutBean" AND NOT "Scale10".QU AND NOT "oSensor3";
   "Scale10".CTU(CU := "mLetOutBean" AND "Clock_0.5Hz" AND NOT "Scale10".QU,
                 R := "iResetCTU",
                 PV := "Mass".Bean,
                 CV => "Weight".Xilo10);
   #_w1 := "mLetOutBean" AND "Scale10".QU;
   "oXilo11" := #_w1 AND NOT "Scale11".QU AND NOT "oSensor3";
   "Scale11".CTU(CU := #_w1 AND "Clock_0.5Hz" AND NOT "Scale11".QU,
                 R := "iResetCTU",
                 PV := "Mass".Bean,
                 CV => "Weight".Xilo11);
   #_w2 := "mLetOutBean" AND "Scale11".QU;
   "oXilo12" := #_w2 AND NOT "Scale12".QU AND NOT "oSensor3";
   "Scale12".CTU(CU := #_w2 AND "Clock_0.5Hz" AND NOT "Scale12".QU,
                 R := "iResetCTU",
                 PV := "Mass".Bean,
                 CV => "Weight".Xilo12);
   "mLightBean" := "Scale12".Q;
END_REGION

REGION Network 8: xả xilo 13,14,15,16 (bột cá)
   // xả xilo 13,14,15,16 (bột cá)
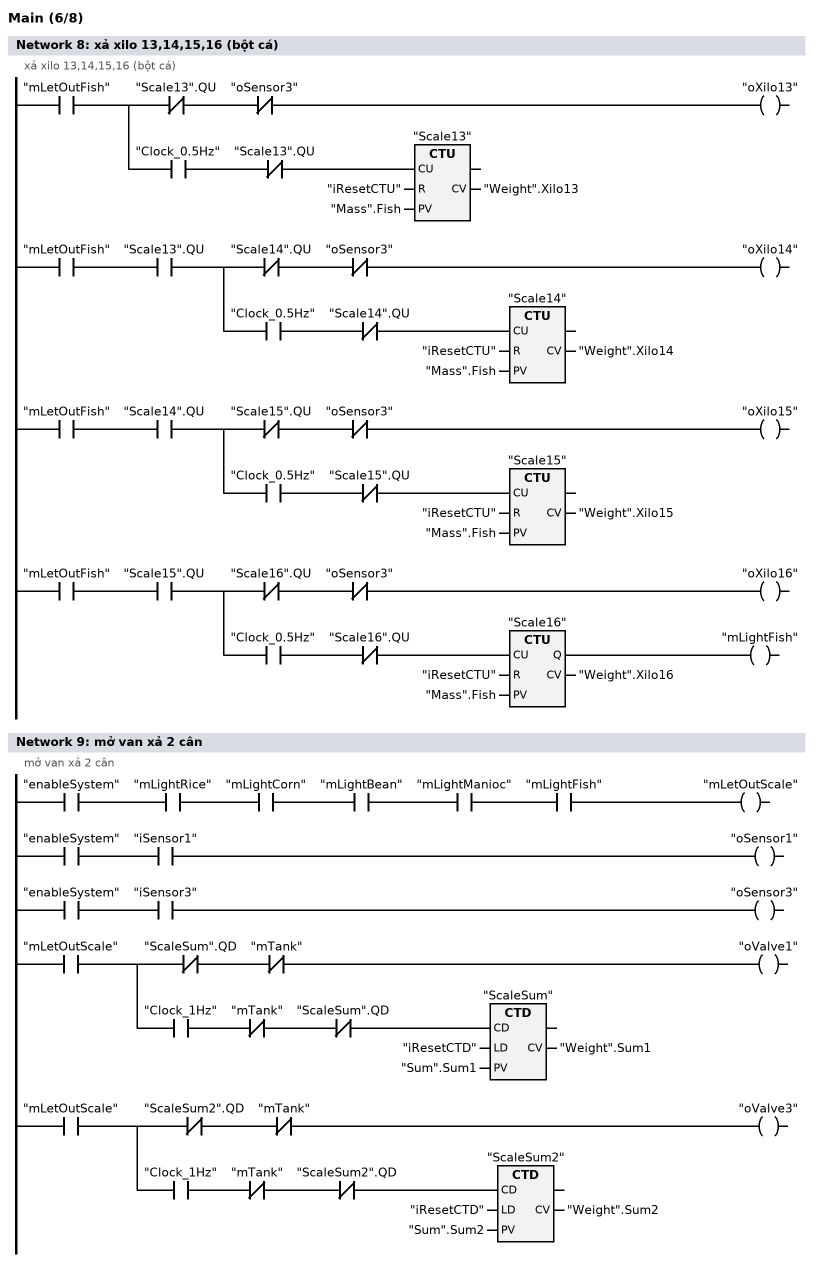
   "oXilo13" := "mLetOutFish" AND NOT "Scale13".QU AND NOT "oSensor3";
   "Scale13".CTU(CU := "mLetOutFish" AND "Clock_0.5Hz" AND NOT "Scale13".QU,
                 R := "iResetCTU",
                 PV := "Mass".Fish,
                 CV => "Weight".Xilo13);
   #_w1 := "mLetOutFish" AND "Scale13".QU;
   "oXilo14" := #_w1 AND NOT "Scale14".QU AND NOT "oSensor3";
   "Scale14".CTU(CU := #_w1 AND "Clock_0.5Hz" AND NOT "Scale14".QU,
                 R := "iResetCTU",
                 PV := "Mass".Fish,
                 CV => "Weight".Xilo14);
   #_w2 := "mLetOutFish" AND "Scale14".QU;
   "oXilo15" := #_w2 AND NOT "Scale15".QU AND NOT "oSensor3";
   "Scale15".CTU(CU := #_w2 AND "Clock_0.5Hz" AND NOT "Scale15".QU,
                 R := "iResetCTU",
                 PV := "Mass".Fish,
                 CV => "Weight".Xilo15);
   #_w3 := "mLetOutFish" AND "Scale15".QU;
   "oXilo16" := #_w3 AND NOT "Scale16".QU AND NOT "oSensor3";
   "Scale16".CTU(CU := #_w3 AND "Clock_0.5Hz" AND NOT "Scale16".QU,
                 R := "iResetCTU",
                 PV := "Mass".Fish,
                 CV => "Weight".Xilo16);
   "mLightFish" := "Scale16".Q;
END_REGION

REGION Network 9: mở van xả 2 cân
   // mở van xả 2 cân
   "mLetOutScale" := "enableSystem" AND "mLightRice" AND "mLightCorn" AND "mLightBean" AND "mLightManioc" AND "mLightFish";
   "oSensor1" := "enableSystem" AND "iSensor1";
   "oSensor3" := "enableSystem" AND "iSensor3";
   "oValve1" := "mLetOutScale" AND NOT "ScaleSum".QD AND NOT "mTank";
   "ScaleSum".CTD(CD := "mLetOutScale" AND "Clock_1Hz" AND NOT "mTank" AND NOT "ScaleSum".QD,
                  LD := "iResetCTD",
                  PV := "Sum".Sum1,
                  CV => "Weight".Sum1);
   "oValve3" := "mLetOutScale" AND NOT "ScaleSum2".QD AND NOT "mTank";
   "ScaleSum2".CTD(CD := "mLetOutScale" AND "Clock_1Hz" AND NOT "mTank" AND NOT "ScaleSum2".QD,
                   LD := "iResetCTD",
                   PV := "Sum".Sum2,
                   CV => "Weight".Sum2);
END_REGION

REGION Network 10: Trộn và xả van 2
   // Trộn và xả van 2
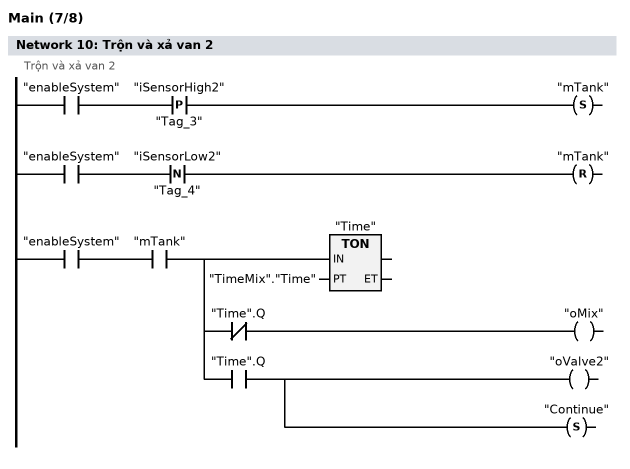
   #_w1 := "enableSystem" AND "iSensorHigh2" AND NOT "Tag_3";   // rising edge of "iSensorHigh2"
   "Tag_3" := "iSensorHigh2";
   IF #_w1 THEN "mTank" := TRUE; END_IF;
   #_w2 := "enableSystem" AND NOT "iSensorLow2" AND "Tag_4";   // falling edge of "iSensorLow2"
   "Tag_4" := "iSensorLow2";
   IF #_w2 THEN "mTank" := FALSE; END_IF;
   #_w3 := "enableSystem" AND "mTank";
   "Time".TON(IN := #_w3, PT := "TimeMix"."Time");
   "oMix" := #_w3 AND NOT "Time".Q;
   "oValve2" := #_w3 AND "Time".Q;
   IF "oValve2" THEN "Continue" := TRUE; END_IF;
END_REGION

REGION Network 11: Hiển thị 2 cân
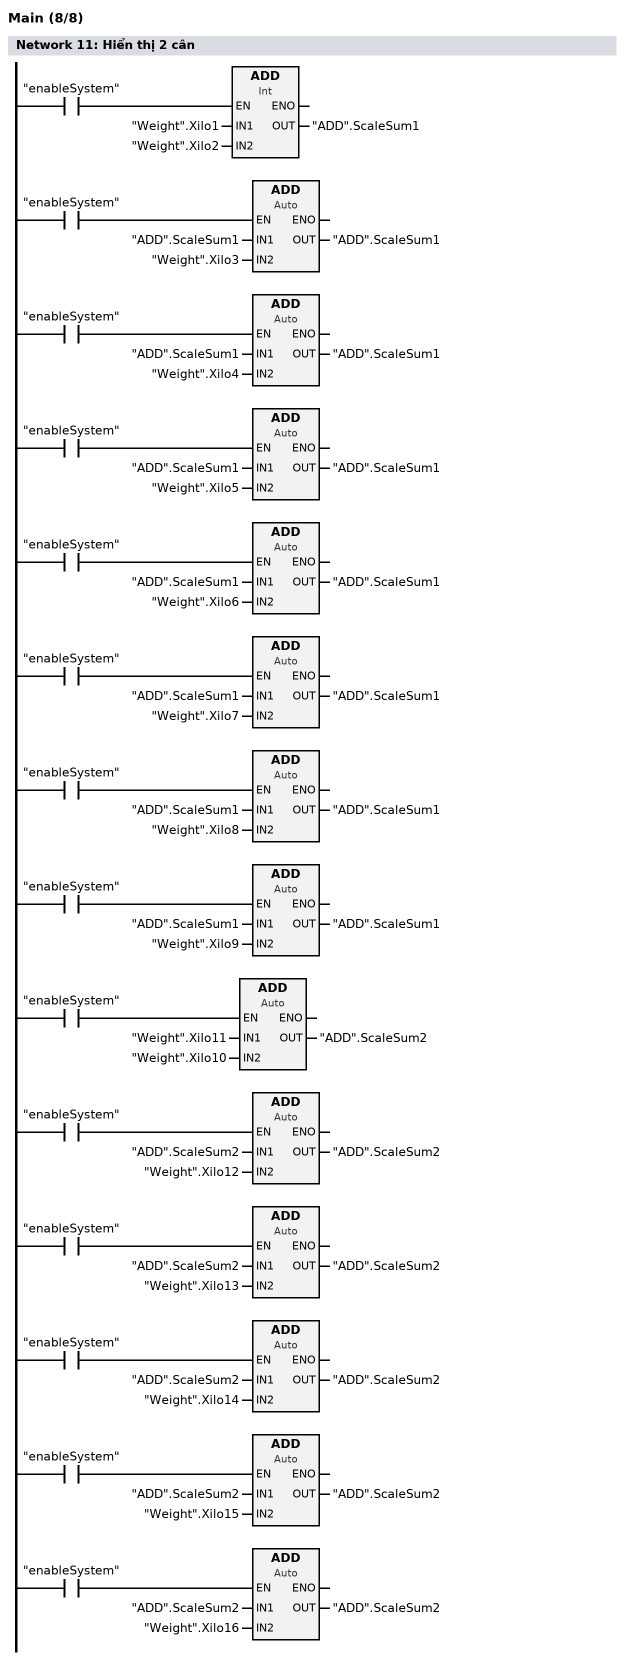
   RUNG wire#powerrail
      Contact( "enableSystem" )
      { S7_Templates := "SrcType := Int" } Add(in1 := "Weight".Xilo1, in2 := "Weight".Xilo2, out => "ADD".ScaleSum1)
   END_RUNG
   RUNG wire#powerrail
      Contact( "enableSystem" )
      Add(in1 := "ADD".ScaleSum1, in2 := "Weight".Xilo3, out => "ADD".ScaleSum1)
   END_RUNG
   RUNG wire#powerrail
      Contact( "enableSystem" )
      Add(in1 := "ADD".ScaleSum1, in2 := "Weight".Xilo4, out => "ADD".ScaleSum1)
   END_RUNG
   RUNG wire#powerrail
      Contact( "enableSystem" )
      Add(in1 := "ADD".ScaleSum1, in2 := "Weight".Xilo5, out => "ADD".ScaleSum1)
   END_RUNG
   RUNG wire#powerrail
      Contact( "enableSystem" )
      Add(in1 := "ADD".ScaleSum1, in2 := "Weight".Xilo6, out => "ADD".ScaleSum1)
   END_RUNG
   RUNG wire#powerrail
      Contact( "enableSystem" )
      Add(in1 := "ADD".ScaleSum1, in2 := "Weight".Xilo7, out => "ADD".ScaleSum1)
   END_RUNG
   RUNG wire#powerrail
      Contact( "enableSystem" )
      Add(in1 := "ADD".ScaleSum1, in2 := "Weight".Xilo8, out => "ADD".ScaleSum1)
   END_RUNG
   RUNG wire#powerrail
      Contact( "enableSystem" )
      Add(in1 := "ADD".ScaleSum1, in2 := "Weight".Xilo9, out => "ADD".ScaleSum1)
   END_RUNG
   RUNG wire#powerrail
      Contact( "enableSystem" )
      Add(in1 := "Weight".Xilo11, in2 := "Weight".Xilo10, out => "ADD".ScaleSum2)
   END_RUNG
   RUNG wire#powerrail
      Contact( "enableSystem" )
      Add(in1 := "ADD".ScaleSum2, in2 := "Weight".Xilo12, out => "ADD".ScaleSum2)
   END_RUNG
   RUNG wire#powerrail
      Contact( "enableSystem" )
      Add(in1 := "ADD".ScaleSum2, in2 := "Weight".Xilo13, out => "ADD".ScaleSum2)
   END_RUNG
   RUNG wire#powerrail
      Contact( "enableSystem" )
      Add(in1 := "ADD".ScaleSum2, in2 := "Weight".Xilo14, out => "ADD".ScaleSum2)
   END_RUNG
   RUNG wire#powerrail
      Contact( "enableSystem" )
      Add(in1 := "ADD".ScaleSum2, in2 := "Weight".Xilo15, out => "ADD".ScaleSum2)
   END_RUNG
   RUNG wire#powerrail
      Contact( "enableSystem" )
      Add(in1 := "ADD".ScaleSum2, in2 := "Weight".Xilo16, out => "ADD".ScaleSum2)
   END_RUNG
   // the same network as SCL:
   IF "enableSystem" THEN
       "ADD".ScaleSum1 := "Weight".Xilo1 + "Weight".Xilo2;
       "ADD".ScaleSum1 := "ADD".ScaleSum1 + "Weight".Xilo3;
       "ADD".ScaleSum1 := "ADD".ScaleSum1 + "Weight".Xilo4;
       "ADD".ScaleSum1 := "ADD".ScaleSum1 + "Weight".Xilo5;
       "ADD".ScaleSum1 := "ADD".ScaleSum1 + "Weight".Xilo6;
       "ADD".ScaleSum1 := "ADD".ScaleSum1 + "Weight".Xilo7;
       "ADD".ScaleSum1 := "ADD".ScaleSum1 + "Weight".Xilo8;
       "ADD".ScaleSum1 := "ADD".ScaleSum1 + "Weight".Xilo9;
       "ADD".ScaleSum2 := "Weight".Xilo11 + "Weight".Xilo10;
       "ADD".ScaleSum2 := "ADD".ScaleSum2 + "Weight".Xilo12;
       "ADD".ScaleSum2 := "ADD".ScaleSum2 + "Weight".Xilo13;
       "ADD".ScaleSum2 := "ADD".ScaleSum2 + "Weight".Xilo14;
       "ADD".ScaleSum2 := "ADD".ScaleSum2 + "Weight".Xilo15;
       "ADD".ScaleSum2 := "ADD".ScaleSum2 + "Weight".Xilo16;
   END_IF;
END_REGION
END_ORGANIZATION_BLOCK